// TIA Portal V20 export
FUNCTION_BLOCK "QDAS_DataManager"   // FB175, LAD
{ S7_Optimized_Access := 'TRUE' }
// stored: IsIECCheckEnabled true, MemoryReserve 100, SetENOAutomatically false
   VAR_INPUT
      reset { ExternalAccessible := 'False'; ExternalVisible := 'False'; ExternalWritable := 'False'} : Bool;
      Trigger { ExternalAccessible := 'False'; ExternalVisible := 'False'; ExternalWritable := 'False'} : Bool;
      readData { ExternalAccessible := 'False'; ExternalVisible := 'False'; ExternalWritable := 'False'} : "typeReadVGageProData";
      reciveBufferData { ExternalAccessible := 'False'; ExternalVisible := 'False'; ExternalWritable := 'False'} : "typeWritePLCData";
   END_VAR
   VAR_OUTPUT
      done { ExternalAccessible := 'False'; ExternalVisible := 'False'; ExternalWritable := 'False'} : Bool;
      occurAlarm { ExternalAccessible := 'False'; ExternalVisible := 'False'; ExternalWritable := 'False'} : Bool;
      sendBufferData { ExternalAccessible := 'False'; ExternalVisible := 'False'; ExternalWritable := 'False'} : "typeReadVGageProData";
      writeData { ExternalAccessible := 'False'; ExternalVisible := 'False'; ExternalWritable := 'False'} : "typeWritePLCData";
   END_VAR
   VAR
      statPLCInputData { ExternalAccessible := 'False'; ExternalVisible := 'False'; ExternalWritable := 'False'} : "typeReadVGageProData";
      statSendCompleted { ExternalAccessible := 'False'; ExternalVisible := 'False'; ExternalWritable := 'False'} : Bool;
      "type" { ExternalAccessible := 'False'; ExternalVisible := 'False'; ExternalWritable := 'False'} : Int;
      module { ExternalAccessible := 'False'; ExternalVisible := 'False'; ExternalWritable := 'False'} : Int;
      machine { ExternalAccessible := 'False'; ExternalVisible := 'False'; ExternalWritable := 'False'} : DInt;
      fixture { ExternalAccessible := 'False'; ExternalVisible := 'False'; ExternalWritable := 'False'} : Int;
      pun { ExternalAccessible := 'False'; ExternalVisible := 'False'; ExternalWritable := 'False'} : Array[0..31] of Char;
      resist { ExternalAccessible := 'False'; ExternalVisible := 'False'; ExternalWritable := 'False'} : Real;
      volt { ExternalAccessible := 'False'; ExternalVisible := 'False'; ExternalWritable := 'False'} : Real;
      current { ExternalAccessible := 'False'; ExternalVisible := 'False'; ExternalWritable := 'False'} : Real;
      instWaitingTimer { ExternalAccessible := 'False'; ExternalVisible := 'False'; ExternalWritable := 'False'} : TON_TIME;
      communicationTimeoutTimer { ExternalAccessible := 'False'; ExternalVisible := 'False'; ExternalWritable := 'False'} : TON_TIME;
      dataDeliveryTimer { ExternalAccessible := 'False'; ExternalVisible := 'False'; ExternalWritable := 'False'} : TON_TIME;
      errCommunicationTimeout { ExternalAccessible := 'False'; ExternalVisible := 'False'; ExternalWritable := 'False'} : Bool;
      errDataDeliveryTimeout { ExternalAccessible := 'False'; ExternalVisible := 'False'; ExternalWritable := 'False'} : Bool;
      detectTrigger { ExternalAccessible := 'False'; ExternalVisible := 'False'; ExternalWritable := 'False'} : Array[0..3] of Bool;
      sequenceTimerStart { ExternalAccessible := 'False'; ExternalVisible := 'False'; ExternalWritable := 'False'} : Bool;
      writeDBWaitTime { ExternalAccessible := 'False'; ExternalVisible := 'False'; ExternalWritable := 'False'} : Time := T#500ms;
   END_VAR
   VAR_TEMP
      tempSendCompletedDefaultData : Bool;
   END_VAR
   VAR CONSTANT
      COMMUNICATION_TIME_OUT_LIMIT : Time := t#10s;
      DELIVERY_TIME_OUT_LIMIT : Time := t#5s;
   END_VAR
   // writeData."type" := 1;
   // writeData.module := 1;
   VAR_TEMP   // added for the SCL form of the ladder/FBD networks
      _w1 : Bool;
      _w2 : Bool;
   END_VAR
BEGIN

REGION Network 1: Check communication
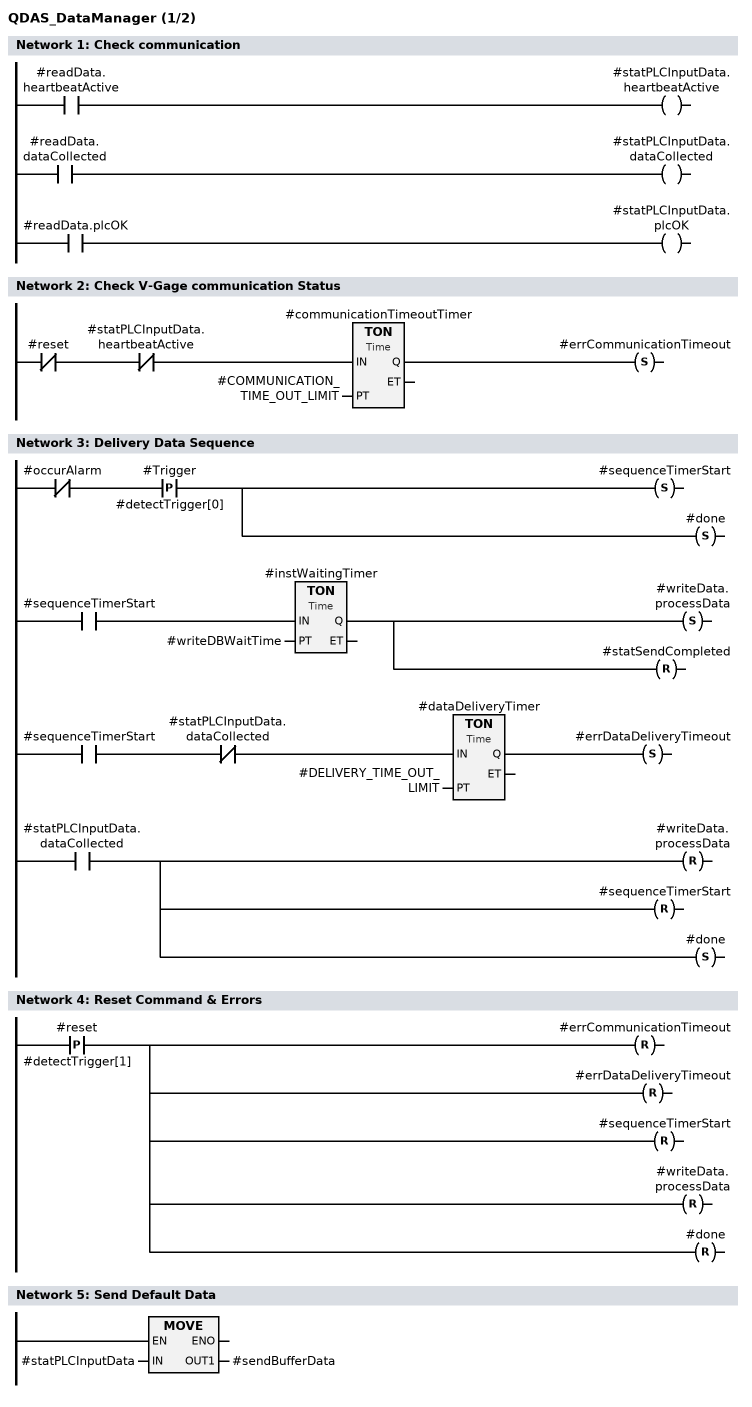
   RUNG wire#powerrail
      Contact( #readData.heartbeatActive )
      Coil( #statPLCInputData.heartbeatActive )
   END_RUNG
   RUNG wire#powerrail
      Contact( #readData.dataCollected )
      Coil( #statPLCInputData.dataCollected )
   END_RUNG
   RUNG wire#powerrail
      Contact( #readData.plcOK )
      Coil( #statPLCInputData.plcOK )
   END_RUNG
   // the same network as SCL:
   #statPLCInputData.heartbeatActive := #readData.heartbeatActive;
   #statPLCInputData.dataCollected := #readData.dataCollected;
   #statPLCInputData.plcOK := #readData.plcOK;
END_REGION

REGION Network 2: Check V-Gage communication Status
   RUNG wire#powerrail
      I_Contact( #reset )
      I_Contact( #statPLCInputData.heartbeatActive )
      { S7_Templates := "time_type := Time" } #communicationTimeoutTimer.TON(pt := #COMMUNICATION_TIME_OUT_LIMIT, et =>)
      S_Coil( #errCommunicationTimeout )
   END_RUNG
   // the same network as SCL:
   #communicationTimeoutTimer(IN := NOT #reset AND NOT #statPLCInputData.heartbeatActive,   // TON
                           PT := #COMMUNICATION_TIME_OUT_LIMIT);
   IF #communicationTimeoutTimer.Q THEN #errCommunicationTimeout := TRUE; END_IF;
END_REGION

REGION Network 3: Delivery Data Sequence
   RUNG wire#powerrail
      I_Contact( #occurAlarm )
      P_Contact(operand := #Trigger, bit := #detectTrigger[0])
      wire#w1
      S_Coil( #sequenceTimerStart )
   END_RUNG
   RUNG wire#w1
      S_Coil( #done )
   END_RUNG
   RUNG wire#powerrail
      Contact( #sequenceTimerStart )
      { S7_Templates := "time_type := Time" } #instWaitingTimer.TON(pt := #writeDBWaitTime, et =>)
      wire#w2
      S_Coil( #writeData.processData )
   END_RUNG
   RUNG wire#w2
      R_Coil( #statSendCompleted )
   END_RUNG
   RUNG wire#powerrail
      Contact( #sequenceTimerStart )
      I_Contact( #statPLCInputData.dataCollected )
      { S7_Templates := "time_type := Time" } #dataDeliveryTimer.TON(pt := #DELIVERY_TIME_OUT_LIMIT, et =>)
      S_Coil( #errDataDeliveryTimeout )
   END_RUNG
   RUNG wire#powerrail
      Contact( #statPLCInputData.dataCollected )
      wire#w3
      R_Coil( #writeData.processData )
   END_RUNG
   RUNG wire#w3
      R_Coil( #sequenceTimerStart )
   END_RUNG
   RUNG wire#w3
      S_Coil( #done )
   END_RUNG
   // the same network as SCL:
   #_w1 := NOT #occurAlarm AND #Trigger AND NOT #detectTrigger[0];   // rising edge of #Trigger
   #detectTrigger[0] := #Trigger;
   IF #_w1 THEN
       #sequenceTimerStart := TRUE;
       #done := TRUE;
   END_IF;
   #instWaitingTimer(IN := #sequenceTimerStart, PT := #writeDBWaitTime);   // TON
   IF #instWaitingTimer.Q THEN
       #writeData.processData := TRUE;
       #statSendCompleted := FALSE;
   END_IF;
   #dataDeliveryTimer(IN := #sequenceTimerStart AND NOT #statPLCInputData.dataCollected,   // TON
                      PT := #DELIVERY_TIME_OUT_LIMIT);
   IF #dataDeliveryTimer.Q THEN #errDataDeliveryTimeout := TRUE; END_IF;
   IF #statPLCInputData.dataCollected THEN
       #writeData.processData := FALSE;
       #sequenceTimerStart := FALSE;
       #done := TRUE;
   END_IF;
END_REGION

REGION Network 4: Reset Command & Errors
   RUNG wire#powerrail
      P_Contact(operand := #reset, bit := #detectTrigger[1])
      wire#w1
      R_Coil( #errCommunicationTimeout )
   END_RUNG
   RUNG wire#w1
      R_Coil( #errDataDeliveryTimeout )
   END_RUNG
   RUNG wire#w1
      R_Coil( #sequenceTimerStart )
   END_RUNG
   RUNG wire#w1
      R_Coil( #writeData.processData )
   END_RUNG
   RUNG wire#w1
      R_Coil( #done )
   END_RUNG
   // the same network as SCL:
   #_w1 := #reset AND NOT #detectTrigger[1];   // rising edge of #reset
   #detectTrigger[1] := #reset;
   IF #_w1 THEN
       #errCommunicationTimeout := FALSE;
       #errDataDeliveryTimeout := FALSE;
       #sequenceTimerStart := FALSE;
       #writeData.processData := FALSE;
       #done := FALSE;
   END_IF;
END_REGION

REGION Network 5: Send Default Data
   RUNG wire#powerrail
      Move(in := #statPLCInputData, out1 => #sendBufferData)
   END_RUNG
   // the same network as SCL:
   #sendBufferData := #statPLCInputData;
END_REGION

REGION Network 6: Write Default Data
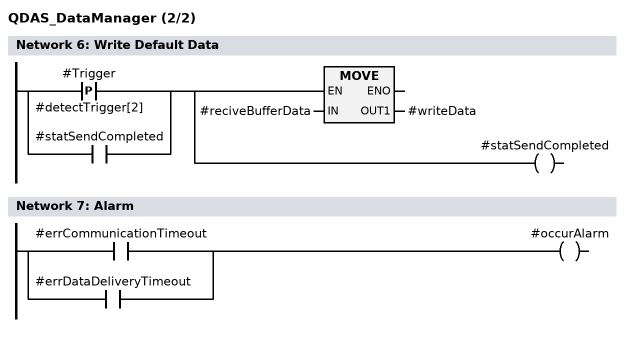
   RUNG wire#powerrail
      P_Contact(operand := #Trigger, bit := #detectTrigger[2])
      wire#w1
      { S7_GenerateENO := "TRUE" } Move(in := #reciveBufferData, out1 => #writeData)
   END_RUNG
   RUNG wire#powerrail
      Contact( #statSendCompleted )
   END_RUNG wire#w1
   RUNG wire#w1
      Coil( #statSendCompleted )
   END_RUNG
   // the same network as SCL:
   #_w1 := #Trigger AND NOT #detectTrigger[2];   // rising edge of #Trigger
   #detectTrigger[2] := #Trigger;
   #_w2 := #_w1 OR #statSendCompleted;
   IF #_w2 THEN #writeData := #reciveBufferData; END_IF;
   #statSendCompleted := #_w2;
END_REGION

REGION Network 7: Alarm
   RUNG wire#powerrail
      Contact( #errCommunicationTimeout )
      wire#w1
      Coil( #occurAlarm )
   END_RUNG
   RUNG wire#powerrail
      Contact( #errDataDeliveryTimeout )
   END_RUNG wire#w1
   // the same network as SCL:
   #occurAlarm := #errCommunicationTimeout OR #errDataDeliveryTimeout;
END_REGION
END_FUNCTION_BLOCK
